TYPE stCBMLInfo :
STRUCT
	sName		: STRING;
	xError 		: BOOL;
	iErrorID 	: INT;
END_STRUCT
END_TYPE

(* stored: Version 1.1.0.1, ProductVersion 3.1.4024.11
   DUT stCBMLInfo: Id {d5a7e22d-2557-45a6-9690-01a82754a23f} *)
